FUNCTION_BLOCK Stereo IMPLEMENTS I_Device
VAR_INPUT
END_VAR
VAR_OUTPUT
END_VAR
VAR
END_VAR

METHOD adjustVolume
ADSLOGSTR(msgCtrlMask := ADSLOG_MSGTYPE_LOG OR ADSLOG_MSGTYPE_LOG,
		msgFmtStr := 'Volume adjusted',
		strArg	:= '');
END_METHOD

{warning 'add method implementation '}
METHOD turnOff
ADSLOGSTR(msgCtrlMask := ADSLOG_MSGTYPE_LOG OR ADSLOG_MSGTYPE_LOG,
		msgFmtStr := 'Stereo is now off',
		strArg	:= '');
END_METHOD

{warning 'add method implementation '}
METHOD turnOn
ADSLOGSTR(msgCtrlMask := ADSLOG_MSGTYPE_LOG OR ADSLOG_MSGTYPE_LOG,
		msgFmtStr := 'Stereo is now on',
		strArg	:= '');
END_METHOD

END_FUNCTION_BLOCK

(* stored: Version 1.1.0.1
   POU Stereo: Id {0ec22f8c-464a-4833-a494-67fc5048899e}, SpecialFunc None
   Method adjustVolume: Id {5e2741da-5aaf-4cc3-bedb-afb5dd6ef0af}
   Method turnOff: Id {d5037d07-130a-4ff4-a8b2-8051332701b7}
   Method turnOn: Id {01af70c0-4843-47f7-9149-beb23180f891} *)
